# EPICS autosave request: softGlueApp/Db/softGlue_FieldIO_descriptions.req
# field I/O descriptions
$(P)$(H)FI1_Signal.DESC
$(P)$(H)FI2_Signal.DESC
$(P)$(H)FI3_Signal.DESC
$(P)$(H)FI4_Signal.DESC
$(P)$(H)FI5_Signal.DESC
$(P)$(H)FI6_Signal.DESC
$(P)$(H)FI7_Signal.DESC
$(P)$(H)FI8_Signal.DESC
$(P)$(H)FI9_Signal.DESC
$(P)$(H)FI10_Signal.DESC
$(P)$(H)FI11_Signal.DESC
$(P)$(H)FI12_Signal.DESC
$(P)$(H)FI13_Signal.DESC
$(P)$(H)FI14_Signal.DESC
$(P)$(H)FI15_Signal.DESC
$(P)$(H)FI16_Signal.DESC
$(P)$(H)FI17_Signal.DESC
$(P)$(H)FI18_Signal.DESC
$(P)$(H)FI19_Signal.DESC
$(P)$(H)FI20_Signal.DESC
$(P)$(H)FI21_Signal.DESC
$(P)$(H)FI22_Signal.DESC
$(P)$(H)FI23_Signal.DESC
$(P)$(H)FI24_Signal.DESC
$(P)$(H)FI25_Signal.DESC
$(P)$(H)FI26_Signal.DESC
$(P)$(H)FI27_Signal.DESC
$(P)$(H)FI28_Signal.DESC
$(P)$(H)FI29_Signal.DESC
$(P)$(H)FI30_Signal.DESC
$(P)$(H)FI31_Signal.DESC
$(P)$(H)FI32_Signal.DESC
$(P)$(H)FI33_Signal.DESC
$(P)$(H)FI34_Signal.DESC
$(P)$(H)FI35_Signal.DESC
$(P)$(H)FI36_Signal.DESC
$(P)$(H)FI37_Signal.DESC
$(P)$(H)FI38_Signal.DESC
$(P)$(H)FI39_Signal.DESC
$(P)$(H)FI40_Signal.DESC
$(P)$(H)FI41_Signal.DESC
$(P)$(H)FI42_Signal.DESC
$(P)$(H)FI43_Signal.DESC
$(P)$(H)FI44_Signal.DESC
$(P)$(H)FI45_Signal.DESC
$(P)$(H)FI46_Signal.DESC
$(P)$(H)FI47_Signal.DESC
$(P)$(H)FI48_Signal.DESC
$(P)$(H)FO1_Signal.DESC
$(P)$(H)FO2_Signal.DESC
$(P)$(H)FO3_Signal.DESC
$(P)$(H)FO4_Signal.DESC
$(P)$(H)FO5_Signal.DESC
$(P)$(H)FO6_Signal.DESC
$(P)$(H)FO7_Signal.DESC
$(P)$(H)FO8_Signal.DESC
$(P)$(H)FO9_Signal.DESC
$(P)$(H)FO10_Signal.DESC
$(P)$(H)FO11_Signal.DESC
$(P)$(H)FO12_Signal.DESC
$(P)$(H)FO13_Signal.DESC
$(P)$(H)FO14_Signal.DESC
$(P)$(H)FO15_Signal.DESC
$(P)$(H)FO16_Signal.DESC
$(P)$(H)FO17_Signal.DESC
$(P)$(H)FO18_Signal.DESC
$(P)$(H)FO19_Signal.DESC
$(P)$(H)FO20_Signal.DESC
$(P)$(H)FO21_Signal.DESC
$(P)$(H)FO22_Signal.DESC
$(P)$(H)FO23_Signal.DESC
$(P)$(H)FO24_Signal.DESC
$(P)$(H)FO25_Signal.DESC
$(P)$(H)FO26_Signal.DESC
$(P)$(H)FO27_Signal.DESC
$(P)$(H)FO28_Signal.DESC
$(P)$(H)FO29_Signal.DESC
$(P)$(H)FO30_Signal.DESC
$(P)$(H)FO31_Signal.DESC
$(P)$(H)FO32_Signal.DESC
$(P)$(H)FO33_Signal.DESC
$(P)$(H)FO34_Signal.DESC
$(P)$(H)FO35_Signal.DESC
$(P)$(H)FO36_Signal.DESC
$(P)$(H)FO37_Signal.DESC
$(P)$(H)FO38_Signal.DESC
$(P)$(H)FO39_Signal.DESC
$(P)$(H)FO40_Signal.DESC
$(P)$(H)FO41_Signal.DESC
$(P)$(H)FO42_Signal.DESC
$(P)$(H)FO43_Signal.DESC
$(P)$(H)FO44_Signal.DESC
$(P)$(H)FO45_Signal.DESC
$(P)$(H)FO46_Signal.DESC
$(P)$(H)FO47_Signal.DESC
$(P)$(H)FO48_Signal.DESC
